FUNCTION sp_input_reducer : real
VAR_INPUT
	sp_auto: REAL;
	sp_manual: REAL;
	sp_tso: REAL;
END_VAR
VAR
END_VAR

sp_input_reducer := 1;

IF GVL.WISNAM_PPC.REMOTE_MODE THEN
	sp_input_reducer := sp_tso;
END_IF


IF GVL.WISNAM_PPC.AUTO_MODE THEN
	IF sp_input_reducer > sp_auto THEN
		sp_input_reducer := sp_auto;
	END_IF
END_IF


IF GVL.WISNAM_PPC.MANUAL_MODE THEN
	IF sp_input_reducer > sp_manual THEN
		sp_input_reducer := sp_manual;
	END_IF
END_IF

END_FUNCTION

(* stored: Version 1.1.0.1, ProductVersion 3.1.4024.15
   POU sp_input_reducer: Id {7c773ba5-11e6-4c53-86be-40a0edacf78a}, SpecialFunc None *)
